// TIA Portal V19 export
TYPE "modTypes"
   STRUCT
      adin { S7_SetPoint := 'True'} : Bool;
      ain { S7_SetPoint := 'True'} : Bool;
      cvlv { S7_SetPoint := 'True'} : Bool;
      din { S7_SetPoint := 'True'} : Bool;
      mtr { S7_SetPoint := 'True'} : Bool;
      mtrDir { S7_SetPoint := 'True'} : Bool;
      mtrLin { S7_SetPoint := 'True'} : Bool;
      vlv { S7_SetPoint := 'True'} : Bool;
   END_STRUCT;
END_TYPE
